# EPICS StreamDevice protocol: devices/devices_drivers/keithley_220/keithley_220.proto
ReplyTimeout = 2000;
InTerminator = CR LF;
ExtraInput = Ignore;

#Set current of K220
setI {
	out "I%fX";
	in"%39c";
}

execute {
	out "X";
	in "%s/NDCI(.*),V.*/";
}

readI {
	out "anythingX";
	in"NDCI%f,V%*f,W%*f,L%*f";
}

readV {
	out "anythingX";
	in"NDCI%*f,V%f,W%*f,L%*f";
}

readW {
	out "anythingX";
	in"NDCI%*f,V%*f,W%f,L%*f";
}

readL {
	out "anythingX";
	in"NDCI%*f,V%*f,W%*f,L%f";
}

readstring {
	out "aX";
	in "%.1/ND(\w\w).*/";
}
